// TIA Portal V19 export
DATA_BLOCK "InfeedPAC3200_AdvMinMax"   // DB37
TITLE = Instance DB of advanced min / max energy data collection
// Instance DB of advanced min / max energy data collection
// stored: InstanceOfName EnS_EnergyDataAdvMinMax, InstanceOfType FB
"EnS_EnergyDataAdvMinMax"
   // VAR_INPUT
   //    advDataMin { ExternalWritable := 'False'} : "EnS_typeEnergyAdv";
   //    advDataMax { ExternalWritable := 'False'} : "EnS_typeEnergyAdv";
   // END_VAR
   // VAR_OUTPUT
   //    error { ExternalAccessible := 'False'; ExternalVisible := 'False'; ExternalWritable := 'False'} : Bool;
   //    status { ExternalAccessible := 'False'; ExternalVisible := 'False'; ExternalWritable := 'False'} : Word;
   // END_VAR
BEGIN
END_DATA_BLOCK
